(* IEC 61131-3 sources: plc_generation_empirical_study/datasets/_archive/pre_native_plcverif_20260810/tasks/C03_E01_forward_reverse_interlock, 2 files *)

(* ---- interface.st ---- *)
FUNCTION_BLOCK C03_E01_forward_reverse_interlock
VAR_INPUT
    ForwardRequest : BOOL;
    ReverseRequest : BOOL;
    Permit : BOOL;
END_VAR
VAR_OUTPUT
    Forward : BOOL;
    Reverse : BOOL;
END_VAR
END_FUNCTION_BLOCK

(* ---- reference.st ---- *)
FUNCTION_BLOCK C03_E01_forward_reverse_interlock
VAR_INPUT
    ForwardRequest : BOOL;
    ReverseRequest : BOOL;
    Permit : BOOL;
END_VAR
VAR_OUTPUT
    Forward : BOOL;
    Reverse : BOOL;
END_VAR

Forward := Permit AND ForwardRequest AND (NOT ReverseRequest);
Reverse := Permit AND ReverseRequest AND (NOT ForwardRequest);

END_FUNCTION_BLOCK
